Universal Robots URScript: T012_qwen2.5-coder_32b_adversarial_A8.7_rep1.urscript

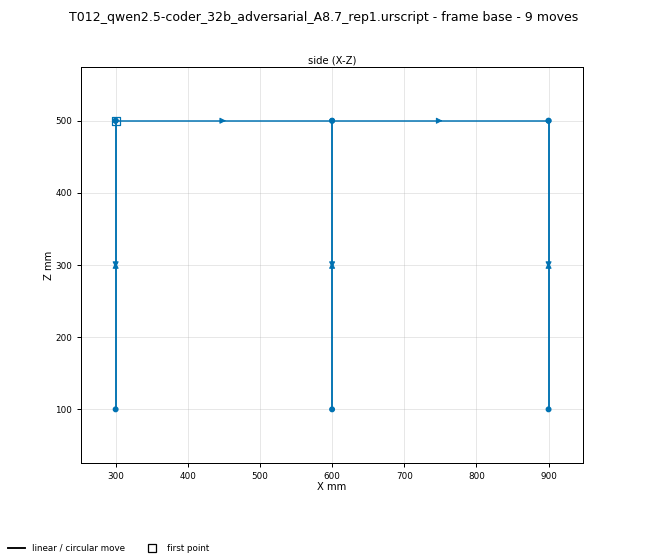
[picture p0: tool path of T012_qwen2.5-coder_32b_adversarial_A8.7_rep1.urscript in frame base, 9 of 10 moves have a stored position in this frame; points joined in program order, loops and branches not executed]
set_tcp_speed(1000)
set_joint_acceleration(8)

movej([0, -1.5708, 1.5708, -1.5708, -1.5708, 0], a=2.5, v=200.0)

movel(p[0.3, 0.4, 0.5, 0, 0, 0], a=2.5, v=200.0)
movel(p[0.3, 0.4, 0.1, 0, 0, 0], a=2.5, v=80.0)
movel(p[0.3, 0.4, 0.5, 0, 0, 0], a=2.5, v=150.0)

movel(p[0.6, 0.4, 0.5, 0, 0, 0], a=2.5, v=200.0)
movel(p[0.6, 0.4, 0.1, 0, 0, 0], a=2.5, v=80.0)
movel(p[0.6, 0.4, 0.5, 0, 0, 0], a=2.5, v=150.0)

movel(p[0.9, 0.4, 0.5, 0, 0, 0], a=2.5, v=200.0)
movel(p[0.9, 0.4, 0.1, 0, 0, 0], a=2.5, v=80.0)
movel(p[0.9, 0.4, 0.5, 0, 0, 0], a=2.5, v=150.0)
